PROGRAM MAIN
VAR
	state		: UINT := 0;
	nextState	: UINT := 0;
	
	mbMaster	: ModbusRtuMaster_KL6x22B;
	mbUnit		: BYTE := 1;
	mbErrorFlag	: BOOL;
	mbErrorId	: MODBUS_ERRORS;
	mbBusy		: BOOL;
	mbBytesRec	: UINT;
	
	mbInputAddr : WORD := 16#D000;
	mbReadAddr	: WORD := 16#D000;
	mbWriteAddr : WORD := 16#D000;
	mbInputData : WORD;
	mbReadData	: WORD;
	mbWriteData : WORD;
	
	inputs		: ARRAY [0..1, 16#00 .. 16#26] OF UINT;
	idx			: WORD;
END_VAR


CASE state OF
0: // init, reset
	FOR idx := 0 TO 16#26 DO
		inputs[0, idx] := 16#D000 + idx;
	END_FOR
	mbInputAddr := 16#D000;
	idx := 0;
	nextState := 1;
	state := 1;

1: // read input registers
	mbMaster.ReadInputRegs(
		UnitID:= mbUnit, 
		Quantity:= 1, 
		MBAddr:= mbInputAddr, 
		cbLength:= SIZEOF(mbInputData), 
		pMemoryAddr:= ADR(mbInputData), 
		Execute:= TRUE, 
		Timeout:= T#1S, 
		BUSY=> mbBusy, 
		Error=> mbErrorFlag, 
		ErrorId=> mbErrorId, 
		cbRead=> mbBytesRec);;

	// if not busy, move to next input register
	IF mbBusy = FALSE THEN
		inputs[1, idx] := mbInputData;
		mbInputAddr := mbInputAddr + 1;
		idx := idx + 1;
		IF idx > 16#26 THEN
			idx := 0;
			mbInputAddr := 16#D000;
		END_IF

		// reset comms and go to next state
		mbMaster.ReadInputRegs(Execute := FALSE);
		state := nextState;
		// catch error
		IF mbErrorFlag = TRUE THEN
			state := 4;
		END_IF
	END_IF
	
2: // read holding register
	mbMaster.ReadRegs(
		UnitID:= mbUnit, 
		Quantity:= 1, 
		MBAddr:= mbReadAddr, 
		cbLength:= SIZEOF(mbReadData), 
		pMemoryAddr:= ADR(mbReadData), 
		Execute:= TRUE, 
		Timeout:= T#1S, 
		BUSY=> mbBusy, 
		Error=> mbErrorFlag, 
		ErrorId=> mbErrorId, 
		cbRead=> mbBytesRec);

	// read complete
	IF mbBusy = FALSE THEN
		// reset comms
		mbMaster.ReadRegs(Execute := FALSE);
		nextState := 1;
		state := nextState;
		// catch error
		IF mbErrorFlag = TRUE THEN
			state := 4;
		END_IF
	END_IF
	
3: // write register
	mbMaster.WriteSingleRegister(
		UnitID:= mbUnit, 
		Quantity:= 1, 
		MBAddr:= mbWriteAddr, 
		cbLength:= SIZEOF(mbWriteData), 
		pMemoryAddr:= ADR(mbWriteData), 
		Execute:= TRUE, 
		Timeout:= T#1S, 
		BUSY=> mbBusy, 
		Error=> mbErrorFlag, 
		ErrorId=> mbErrorId, 
		cbRead=> mbBytesRec);

	// write complete
	IF mbBusy = FALSE THEN
		// reset comms
		mbMaster.ReadRegs(Execute := FALSE);
		nextState := 1;
		state := nextState;
		// catch error
		IF mbErrorFlag = TRUE THEN
			state := 4;
		END_IF
	END_IF

4: // error, wait for reset

ELSE // stop
	
END_CASE

END_PROGRAM

(* stored: Version 1.1.0.1, ProductVersion 3.1.4024.6
   POU MAIN: Id {7212b5d2-df33-4916-8615-e5304be4440a}, SpecialFunc None *)
